FUNCTION FUN_get_Posicion_Ocupada_Array : INT
VAR_INPUT
	color : INT;
END_VAR
VAR
	i 				: INT;
	ContadorPalets 	: INT  := 0;
	ocupada 		: BOOL := TRUE;	
END_VAR


// Retorna la primera posicion ocupada del color correspondiente en el array Clasificados
FOR i := 0 TO 53 DO
	IF GVL.Clasificados[i].Color = color THEN
		ContadorPalets := ContadorPalets +1;
		IF ocupada THEN
			FUN_get_Posicion_Ocupada_Array := i+1;
			ocupada := FALSE;
		END_IF
	END_IF
END_FOR

IF ocupada THEN
	FUN_get_Posicion_Ocupada_Array := 0;
END_IF

GVL.ContadorPalets := ContadorPalets;

END_FUNCTION

(* stored: Version 1.1.0.1, ProductVersion 3.1.4024.12
   POU FUN_get_Posicion_Ocupada_Array: Id {91a977c7-2f6f-4f75-97f3-ed700e87417d}, SpecialFunc None *)
